INTERFACE I_SerialByteConnection

PROPERTY ByteData : BYTE
GET
END_GET
END_PROPERTY

PROPERTY ByteDataRecieved : BOOL
GET
END_GET
END_PROPERTY

METHOD SendAByte : HRESULT
VAR_INPUT
	DataToSend : BYTE;
END_VAR
END_METHOD

END_INTERFACE

(* stored: Version 1.1.0.1, ProductVersion 3.1.4026.18
   Itf I_SerialByteConnection: Id {00a5bad9-6763-42c4-8902-f64c5ba333d5}
   Property ByteData: Id {656f7cd0-c916-4807-9bdf-77f84d9beb68}
   Get Get: Id {033eef38-8531-4af4-842a-ae03fdfb9840}
   Property ByteDataRecieved: Id {58fc521f-68b7-46c0-b15a-31f40e325f44}
   Get Get: Id {439accd9-8dd1-4931-a322-c6a097c0005f}
   Method SendAByte: Id {4dd28dde-0709-4ab0-8d33-eb2cf7c91d2a} *)
